(* PLC project Sin nombre, Desconocido Sin nombre 1 *)
(* stored: creationDateTime 2024-10-23T14:22:18, modificationDateTime 2024-10-24T11:30:04 *)

PROGRAM program0s
  VAR
    sensor AT %IW0.0 : UINT := 0;
  END_VAR
  VAR CONSTANT
    min_baj : UINT := 33400;
  END_VAR
  VAR
    luz AT %QX0.0 : BOOL := 0;
    luz1 AT %QX0.1 : BOOL := 0;
  END_VAR
  VAR CONSTANT
    min_ALT : UINT := 34501;
    min_sup : UINT := 36801;
    tope_baj : UINT := 34500;
    tope_alt : UINT := 36800;
    tope_sup : UINT := 38400;
  END_VAR
  VAR
    acum : UINT := 0;
    timer_normal : BOOL := 1;
    timer_alt : BOOL := 0;
    timer_sup : BOOL := 0;
    probarSup : BOOL := 0;
    probarNorm : BOOL := 0;
    ProbarAlt : BOOL := 0;
    inicio : BOOL := 0;
    TON0 : TON;
    CTU_LINT0 : CTU_LINT;
    CTU_LINT1 : CTU_LINT;
    TON1 : TON;
    CTU_LINT2 : CTU_LINT;
  END_VAR
  VAR  (* added by the conversion: wires and edge detectors of the diagram *)
    R_TRIG1 : R_TRIG;
    _GE109_ENO : BOOL;
    _GE109_OUT : BOOL;
    _NOT120_OUT : BOOL;
    _ADD105_ENO : BOOL;
    _ADD105_OUT : UINT;
    R_TRIG2 : R_TRIG;
    _GE2_ENO : BOOL;
    _GE2_OUT : BOOL;
    _ADD9_ENO : BOOL;
    _ADD9_OUT : UINT;
    R_TRIG3 : R_TRIG;
    _LE124_ENO : BOOL;
    _LE124_OUT : BOOL;
  END_VAR

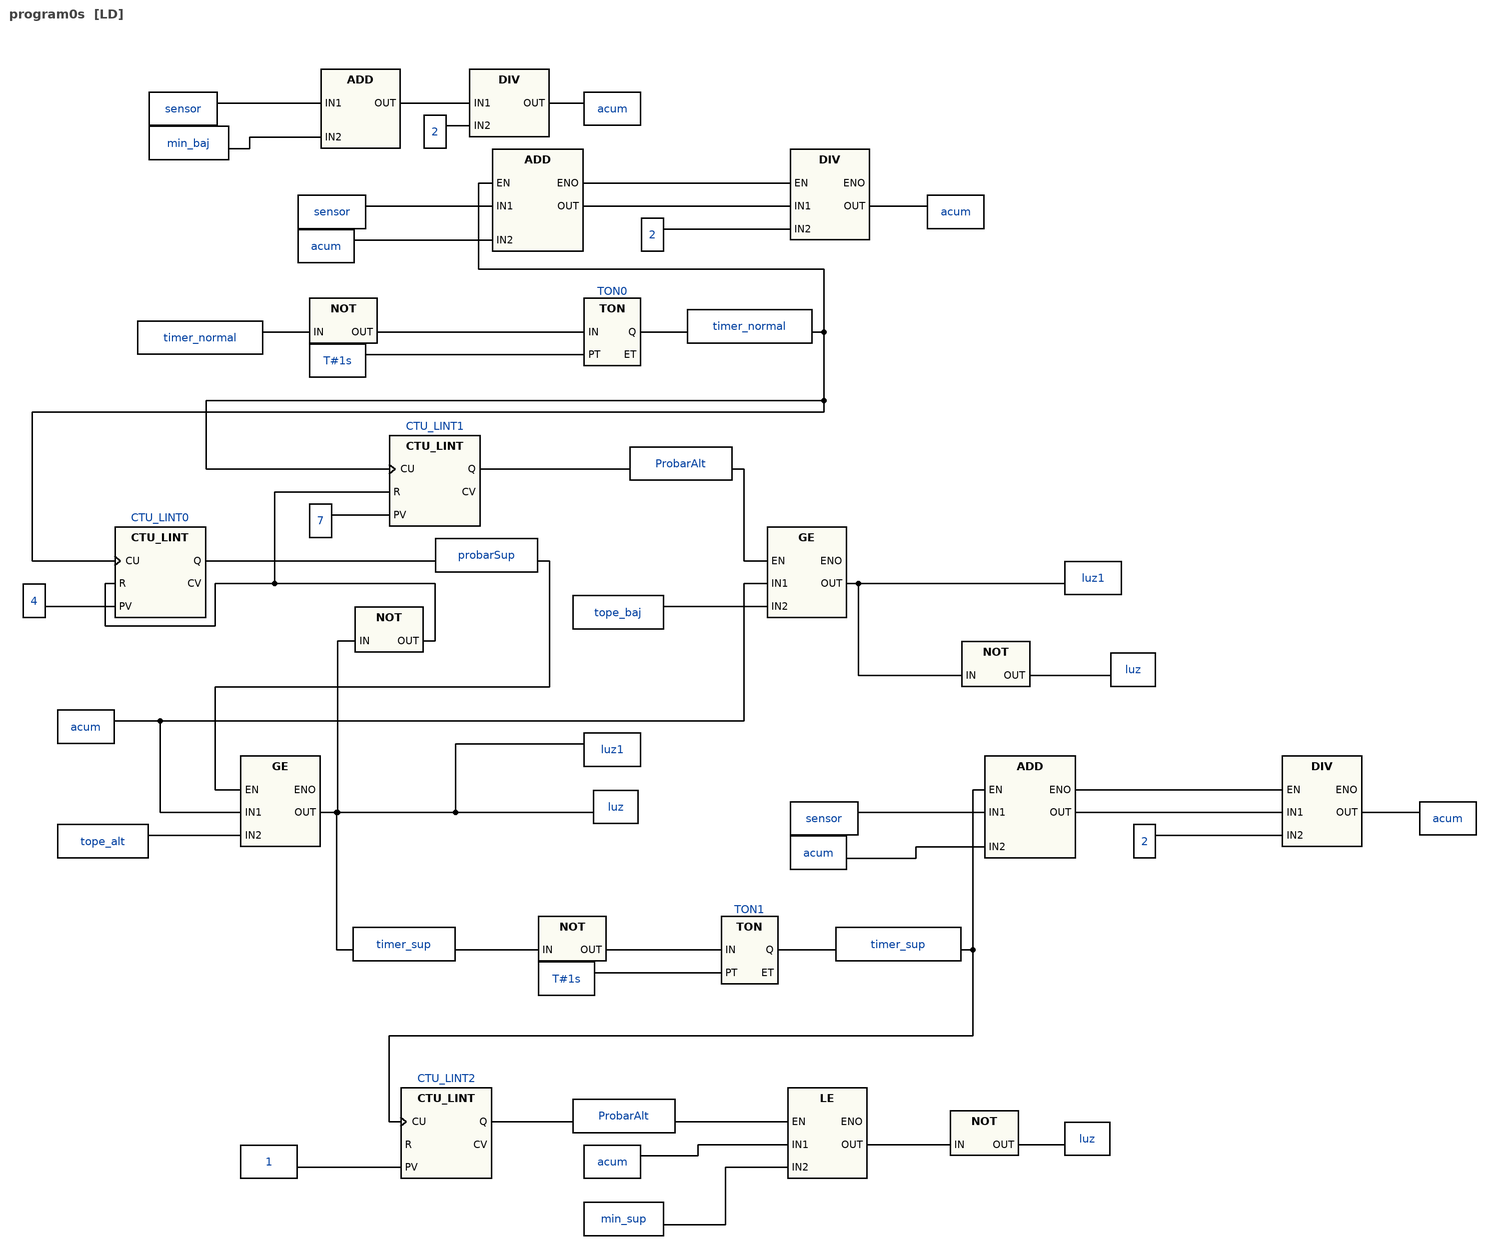
(* LD diagram, written out as Structured Text *)
acum := (sensor + min_baj) / 2;
TON0(IN := NOT timer_normal, PT := T#1s);
timer_normal := TON0.Q;
R_TRIG1(CLK := timer_normal);
_GE109_OUT := GE(EN := probarSup, IN1 := acum, IN2 := tope_alt, ENO => _GE109_ENO);
_NOT120_OUT := NOT _GE109_OUT;
CTU_LINT0(CU := R_TRIG1.Q, R := _NOT120_OUT, PV := 4);
probarSup := CTU_LINT0.Q;
_ADD105_OUT := ADD(EN := timer_normal, IN1 := sensor, IN2 := acum, ENO => _ADD105_ENO);
IF _ADD105_ENO THEN acum := _ADD105_OUT / 2; END_IF;
IF _GE109_ENO THEN luz := _GE109_OUT; END_IF;
IF _GE109_ENO THEN luz1 := _GE109_OUT; END_IF;
R_TRIG2(CLK := timer_normal);
CTU_LINT1(CU := R_TRIG2.Q, R := _NOT120_OUT, PV := 7);
ProbarAlt := CTU_LINT1.Q;
_GE2_OUT := GE(EN := ProbarAlt, IN1 := acum, IN2 := tope_baj, ENO => _GE2_ENO);
IF _GE2_ENO THEN luz1 := _GE2_OUT; END_IF;
luz := NOT _GE2_OUT;
IF _GE109_ENO THEN timer_sup := _GE109_OUT; END_IF;
TON1(IN := NOT timer_sup, PT := T#1s);
timer_sup := TON1.Q;
_ADD9_OUT := ADD(EN := timer_sup, IN1 := sensor, IN2 := acum, ENO => _ADD9_ENO);
IF _ADD9_ENO THEN acum := _ADD9_OUT / 2; END_IF;
R_TRIG3(CLK := timer_sup);
CTU_LINT2(CU := R_TRIG3.Q, PV := 1);
ProbarAlt := CTU_LINT2.Q;
_LE124_OUT := LE(EN := ProbarAlt, IN1 := acum, IN2 := min_sup, ENO => _LE124_ENO);
luz := NOT _LE124_OUT;
END_PROGRAM

CONFIGURATION Config0
  RESOURCE Res0 ON PLC
    TASK task0(INTERVAL := T#20ms, PRIORITY := 0);
    PROGRAM instance0 WITH task0 : program0s;
  END_RESOURCE
END_CONFIGURATION
